# EPICS alarm handler configuration: alh_files/mgnt_li25.alhConfig
GROUP NULL MGNT:LI25:1
   $COMMAND edm -x -eolc -noedit mgnt_li25_main.edl

$ALIAS LI25
$GUIDANCE
li25 Magnets
   Group Name: MGNT:LI25:1
   Summary PV:  MGNT:LI25:1:STATSUMY
$END

   INCLUDE MGNT:LI25:1 ./mgnt_li25_kick.alhConfig
   INCLUDE MGNT:LI25:1 ./mgnt_li25_lgps.alhConfig
   INCLUDE MGNT:LI25:1 ./mgnt_li25_quad.alhConfig
   INCLUDE MGNT:LI25:1 ./mgnt_li25_xcor.alhConfig
   INCLUDE MGNT:LI25:1 ./mgnt_li25_ycor.alhConfig
